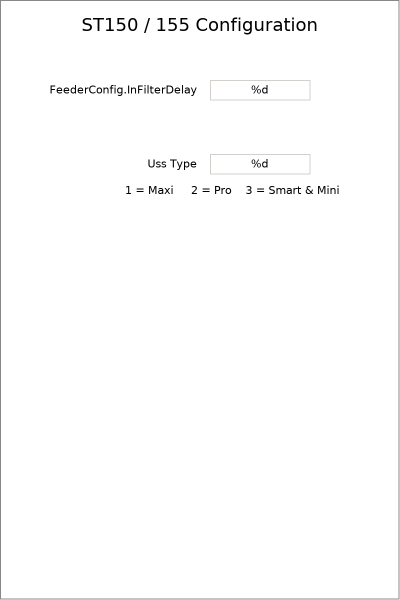
VISUALIZATION VISU_Recipe_ST160  // 400x600
    Textfield (210,80 100x20), "%d", text variable: _20_AUTO.recipe.st150.USS_ErrorTime_ms
        OnMouseDown: write the text variable via Default
    Label (0,5 400x40), "ST150 / 155 Configuration"
    Label (0,80 200x20), "FeederConfig.InFilterDelay"
    Textfield (210,154 100x20), "%d", text variable: _20_AUTO.recipe.st150.USS_Type
        OnMouseDown: write the text variable via Default
    Label (0,154 200x20), "Uss Type"
    Label (112,176 241x29), "1 = Maxi 2 = Pro 3 = Smart & Mini"
END_VISUALIZATION

(* stored: Version 1.1.0.1, ProductVersion 3.1.4024.6
   Visu VISU_Recipe_ST160: Id {cedf75af-695d-41a6-86be-517076040af4} *)
